PROGRAM MAIN
VAR
END_VAR

Comandi();
Motore();

ACTION Comandi:
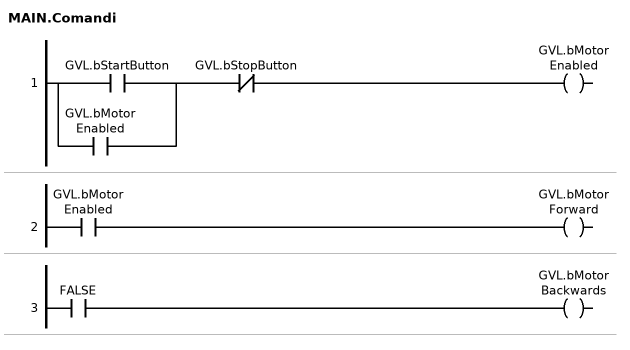
// NETWORK 1
GVL.bMotorEnabled := (GVL.bStartButton OR GVL.bMotorEnabled) AND NOT GVL.bStopButton;

// NETWORK 2
GVL.bMotorForward := GVL.bMotorEnabled;

// NETWORK 3
GVL.bMotorBackwards := FALSE;
END_ACTION

ACTION Motore:
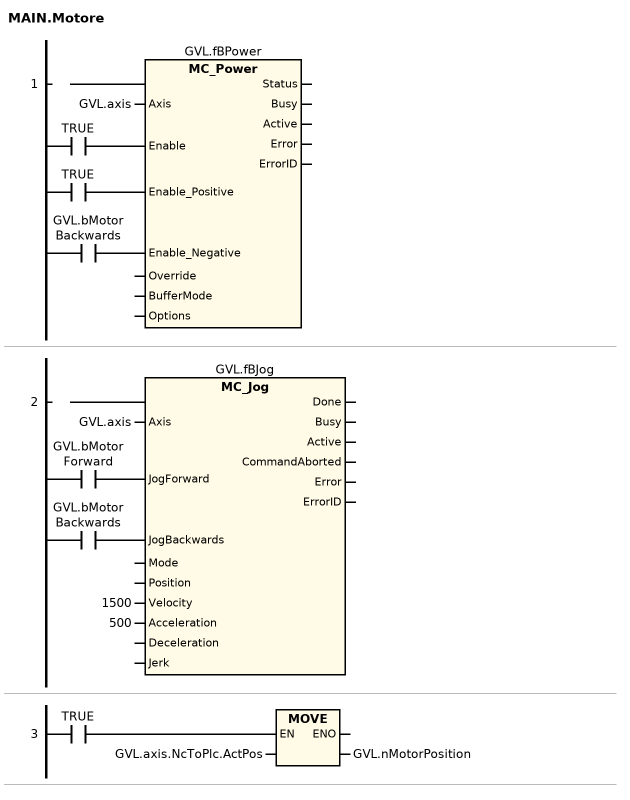
// NETWORK 1
GVL.fBPower(
    Axis := GVL.axis,
    Enable := TRUE,
    Enable_Positive := TRUE,
    Enable_Negative := GVL.bMotorBackwards); // MC_Power

// NETWORK 2
GVL.fBJog(
    Axis := GVL.axis,
    JogForward := GVL.bMotorForward,
    JogBackwards := GVL.bMotorBackwards,
    Velocity := 1500,
    Acceleration := 500); // MC_Jog

// NETWORK 3
GVL.nMotorPosition := GVL.axis.NcToPlc.ActPos;
END_ACTION

END_PROGRAM

(* stored: Version 1.1.0.1, ProductVersion 3.1.4024.12
   POU MAIN: Id {f15a0d18-3609-45db-8199-b71f90c9c6f3}, SpecialFunc None
   Action Comandi: Id {58a29216-9b6a-4898-a724-3758db858095}
   Action Motore: Id {097a3c3a-5458-406a-9471-0adcefc77b8a} *)
